TYPE ST_InputVoltageMeter :
STRUCT
	GenPhaseVoltage : ARRAY[1..3] OF REAL;
	GenLineVoltage : ARRAY[1..3] OF REAL;
	GenFrequency : REAL;
	GenFieldDirection: BOOL;
	EL3443Status	:	UINT;
END_STRUCT
END_TYPE

(* stored: Version 1.1.0.1, ProductVersion 3.1.4024.12
   DUT ST_InputVoltageMeter: Id {de58f2c8-ab7e-4ca9-b3b6-48b1f814e6fb} *)
